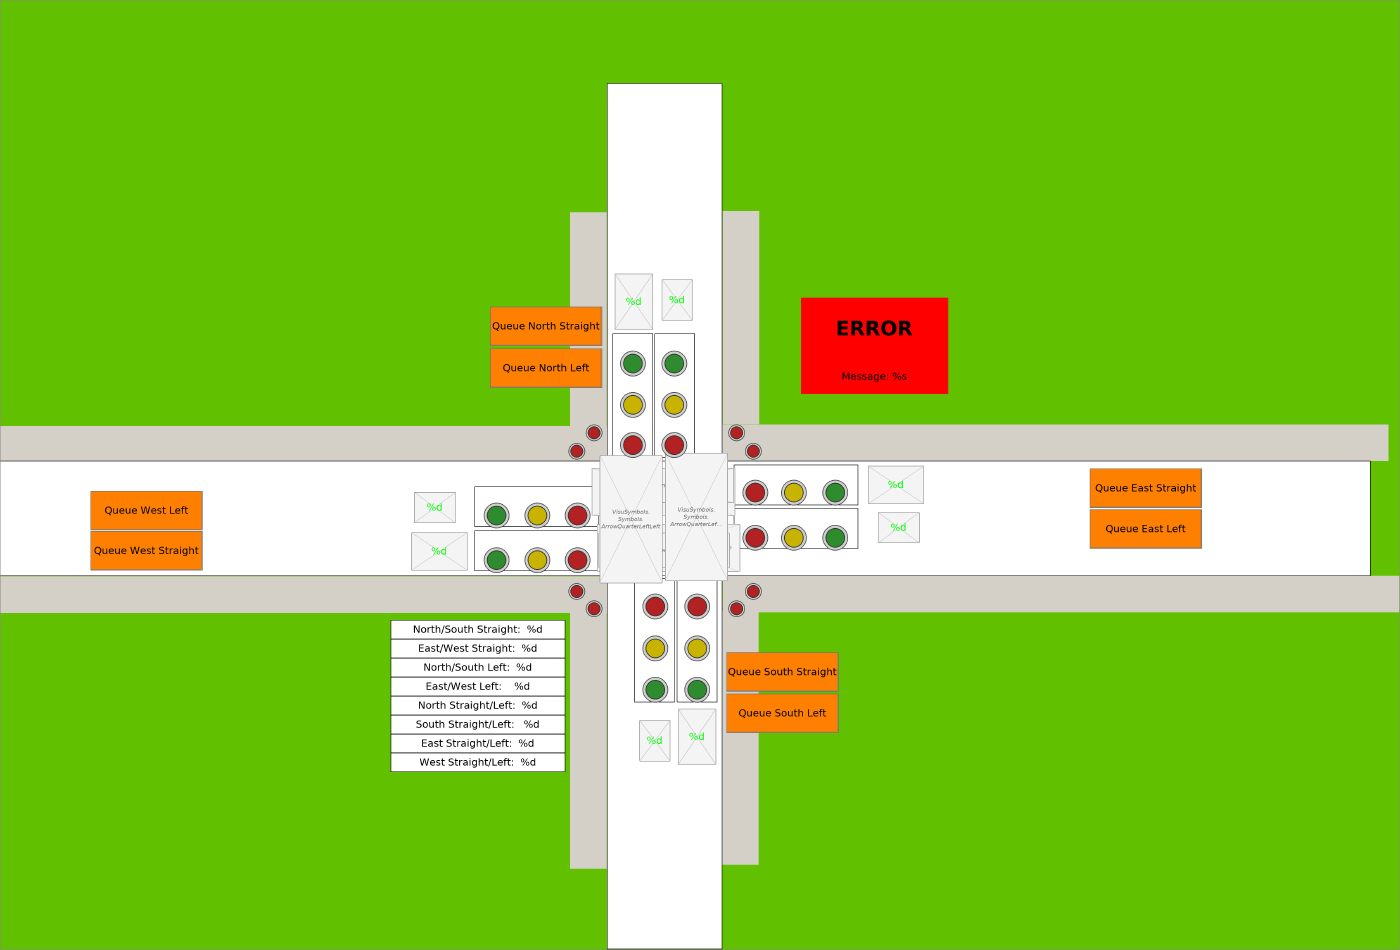
VISUALIZATION IntersectionVisual  // 2505x1701
    Rectangle (1292,1094 65x454)
    Rectangle (1020,1095 65x460)
    Rectangle (1020,380 65x384)
    Rectangle (1293,378 65x381)
    Rectangle (1293,1031 1210x65)
    Rectangle (0,1032 1088x65)
    Rectangle (0,763 1086x65)
    Rectangle (1291,760 1193x65)
    Rectangle (1086,149 206x1550)
    Rectangle (0,825 2452x206)
    Label (2086,901 197x64), "East"
    Label (1090,415 197x64), "North"
    Label (1091,1392 197x64), "South"
    Label (14,891 197x64), "West"
    RoundedRectangle (1313,832 222x72)
    Lamp1 (1394,840 53x84), variable: EastLight_Control.StraightYellowLight, style: Lamp-Lamp1-Yellow
    Lamp1 (1468,840 53x84), variable: EastLight_Control.StraightGreenLight, style: Lamp-Lamp1-Green
    Image (1553,834 100x68), "%d", text variable: Glbl.eastStraightSensorCnt, invisible if: NOT Glbl.eastStraightSensor, image: VisuSymbols.Symbols.ArrowBoldLeft
    RoundedRectangle (1313,910 222x72)
    Lamp1 (1394,921 53x84), variable: EastLight_Control.LeftYellowLight, style: Lamp-Lamp1-Yellow
    Lamp1 (1468,921 53x84), variable: EastLight_Control.LeftGreenLight, style: Lamp-Lamp1-Green
    Image (1571,917 74x55), "%d", text variable: Glbl.eastLeftSensorCnt, colour toggle: Glbl.eastLeftSensor, invisible if: Not Glbl.eastLeftSensor, image: VisuSymbols.Symbols.ArrowBoldDown
    Button (1950,839 200x70), "Queue East Straight"
        OnMouseDown: execute { Glbl.eastStraightSensor := TRUE; Glbl.eastStraightSensorCnt := Glbl.eastStraightSensorCnt + 1; }
    Button (1950,912 200x70), "Queue East Left"
        OnMouseDown: execute { Glbl.eastLeftSensor := TRUE; Glbl.eastLeftSensorCnt := Glbl.eastLeftSensorCnt + 1; }
    RoundedRectangle (849,871 222x72)
    RoundedRectangle (849,950 222x72)
    Lamp1 (1007,881 53x84), variable: WestLight_Control.LeftRedLight, style: Lamp-Lamp1-Red
    Lamp1 (935,881 53x84), variable: WestLight_Control.LeftYellowLight, style: Lamp-Lamp1-Yellow
    Lamp1 (862,881 53x84), variable: WestLight_Control.LeftGreenLight, style: Lamp-Lamp1-Green
    Lamp1 (1007,961 53x84), variable: WestLight_Control.StraightRedLight, style: Lamp-Lamp1-Red
    Lamp1 (935,961 53x84), variable: WestLight_Control.StraightYellowLight, style: Lamp-Lamp1-Yellow
    Lamp1 (862,961 53x84), variable: WestLight_Control.StraightGreenLight, style: Lamp-Lamp1-Green
    Image (736,953 100x68), "%d", text variable: Glbl.westStraightSensorCnt, invisible if: Not Glbl.westStraightSensor, image: VisuSymbols.Symbols.ArrowBoldRight
    Image (741,881 74x55), "%d", text variable: Glbl.westLeftSensorCnt, invisible if: Not Glbl.westLeftSensor, image: VisuSymbols.Symbols.ArrowBoldUp
    Button (162,951 200x70), "Queue West Straight"
        OnMouseDown: execute { Glbl.westStraightSensor := TRUE; Glbl.westStraightSensorCnt := Glbl.westStraightSensorCnt + 1; }
    Button (162,879 200x70), "Queue West Left"
        OnMouseDown: execute { Glbl.westLeftSensor := TRUE; Glbl.westLeftSensorCnt := Glbl.westLeftSensorCnt + 1; }
    Lamp1 (1301,1070 34x40), variable: SouthLight_Control.CrosswalkLight, invisible if: NOT SouthLight_Control.CrosswalkLight, style: Lamp-Lamp1-Green
    Lamp1 (1331,1039 34x40), variable: EastLight_Control.CrosswalkLight, invisible if: NOT EastLight_Control.CrosswalkLight, style: Lamp-Lamp1-Green
    Lamp1 (1046,1070 34x40), variable: SouthLight_Control.CrosswalkLight, invisible if: NOT SouthLight_Control.CrosswalkLight, style: Lamp-Lamp1-Green
    Lamp1 (1015,1039 34x40), variable: WestLight_Control.CrosswalkLight, invisible if: NOT WestLight_Control.CrosswalkLight, style: Lamp-Lamp1-Green
    Lamp1 (1331,788 34x40), variable: EastLight_Control.CrosswalkLight, invisible if: NOT EastLight_Control.CrosswalkLight, style: Lamp-Lamp1-Green
    Lamp1 (1301,755 34x40), variable: NorthLight_Control.CrosswalkLight, invisible if: NOT NorthLight_Control.CrosswalkLight, style: Lamp-Lamp1-Green
    Lamp1 (1015,788 34x40), variable: WestLight_Control.CrosswalkLight, invisible if: NOT WestLight_Control.CrosswalkLight, style: Lamp-Lamp1-Green
    Lamp1 (1046,755 34x40), variable: NorthLight_Control.CrosswalkLight, invisible if: NOT NorthLight_Control.CrosswalkLight, style: Lamp-Lamp1-Green
    Lamp1 (1331,788 34x40), variable: NOT EastLight_Control.CrosswalkLight, invisible if: EastLight_Control.CrosswalkLight, style: Lamp-Lamp1-Red
    Lamp1 (1301,755 34x40), variable: NOT NorthLight_Control.CrosswalkLight, invisible if: NorthLight_Control.CrosswalkLight, style: Lamp-Lamp1-Red
    Lamp1 (1331,1039 34x40), variable: NOT EastLight_Control.CrosswalkLight, invisible if: EastLight_Control.CrosswalkLight, style: Lamp-Lamp1-Red
    Lamp1 (1301,1070 34x40), variable: NOT SouthLight_Control.CrosswalkLight, invisible if: SouthLight_Control.CrosswalkLight, style: Lamp-Lamp1-Red
    Lamp1 (1046,755 34x40), variable: NOT NorthLight_Control.CrosswalkLight, invisible if: NorthLight_Control.CrosswalkLight, style: Lamp-Lamp1-Red
    Lamp1 (1015,788 34x40), variable: NOT WestLight_Control.CrosswalkLight, invisible if: WestLight_Control.CrosswalkLight, style: Lamp-Lamp1-Red
    Lamp1 (1015,1039 34x40), variable: NOT WestLight_Control.CrosswalkLight, invisible if: WestLight_Control.CrosswalkLight, style: Lamp-Lamp1-Red
    Lamp1 (1046,1070 34x40), variable: NOT SouthLight_Control.CrosswalkLight, invisible if: SouthLight_Control.CrosswalkLight, style: Lamp-Lamp1-Red
    Image (1059,838 256x85), invisible if: NOT Glbl.westLeftActive, image: VisuSymbols.Symbols.ArrowQuarterLeftUp
    Image (1068,938 256x85), invisible if: NOT Glbl.eastLeftActive, image: VisuSymbols.Symbols.ArrowQuarterLeftDown
    Image (1079,838 234x62), invisible if: NOT Glbl.eastStraightActive, image: VisuSymbols.Symbols.ArrowBoldLeft
    Image (1071,954 234x62), invisible if: Not Glbl.westStraightActive, image: VisuSymbols.Symbols.ArrowBoldRight
    RoundedRectangle (1211,1035 72x222)
    RoundedRectangle (1135,1035 72x222)
    Lamp1 (1221,1044 53x84), variable: SouthLight_Control.StraightRedLight, style: Lamp-Lamp1-Red
    Lamp1 (1146,1044 53x84), variable: SouthLight_Control.LeftRedLight, style: Lamp-Lamp1-Red
    Lamp1 (1146,1119 53x84), variable: SouthLight_Control.LeftYellowLight, style: Lamp-Lamp1-Yellow
    Lamp1 (1221,1119 53x84), variable: SouthLight_Control.StraightYellowLight, style: Lamp-Lamp1-Yellow
    Lamp1 (1146,1193 53x84), variable: SouthLight_Control.LeftGreenLight, style: Lamp-Lamp1-Green
    Lamp1 (1221,1193 53x84), variable: SouthLight_Control.StraightGreenLight, style: Lamp-Lamp1-Green
    Button (1300,1168 200x70), "Queue South Straight"
        OnMouseDown: execute { Glbl.southStraightSensor := TRUE; Glbl.southStraightSensorCnt := Glbl.southStraightSensorCnt + 1; }
    Button (1300,1242 200x70), "Queue South Left"
        OnMouseDown: execute { Glbl.southLeftSensor := TRUE; Glbl.southLeftSensorCnt := Glbl.southLeftSensorCnt + 1; }
    RoundedRectangle (1096,597 72x222)
    RoundedRectangle (1171,597 72x222)
    Image (1144,1289 55x74), "%d", text variable: Glbl.southLeftSensorCnt, invisible if: NOT Glbl.southLeftSensor, image: VisuSymbols.Symbols.ArrowBoldLeft
    Image (1213,1269 68x100), "%d", text variable: Glbl.southStraightSensorCnt, invisible if: Not Glbl.southStraightSensor, image: VisuSymbols.Symbols.ArrowBoldUp
    Image (1096,822 62x193), colour toggle: Glbl.eastLeftSensor, invisible if: Not Glbl.northStraightActive, image: VisuSymbols.Symbols.ArrowBoldDown
    Image (1215,841 62x193), invisible if: Not Glbl.southStraightActive, image: VisuSymbols.Symbols.ArrowBoldUp
    Image (1190,811 112x229), invisible if: NOT Glbl.northLeftActive, image: VisuSymbols.Symbols.ArrowQuarterLeftRight
    Image (1073,815 112x229), invisible if: NOT Glbl.southLeftActive, image: VisuSymbols.Symbols.ArrowQuarterLeftLeft
    Lamp1 (1106,755 53x84), variable: NorthLight_Control.StraightRedLight, style: Lamp-Lamp1-Red
    Lamp1 (1106,683 53x84), variable: NorthLight_Control.StraightYellowLight, style: Lamp-Lamp1-Yellow
    Lamp1 (1106,609 53x84), variable: NorthLight_Control.StraightGreenLight, style: Lamp-Lamp1-Green
    Lamp1 (1180,755 53x84), variable: NorthLight_Control.LeftRedLight, style: Lamp-Lamp1-Red
    Lamp1 (1180,683 53x84), variable: NorthLight_Control.LeftYellowLight, style: Lamp-Lamp1-Yellow
    Lamp1 (1180,609 53x84), variable: NorthLight_Control.LeftGreenLight, style: Lamp-Lamp1-Green
    Button (877,549 200x70), "Queue North Straight"
        OnMouseDown: execute { Glbl.northStraightSensor := TRUE; Glbl.northStraightSensorCnt := Glbl.northStraightSensorCnt + 1; }
    Button (877,624 200x70), "Queue North Left"
        OnMouseDown: execute { Glbl.northLeftSensor := TRUE; Glbl.northLeftSensorCnt := Glbl.northLeftSensorCnt + 1; }
    Image (1100,490 68x100), "%d", text variable: Glbl.northStraightSensorCnt, colour toggle: Glbl.eastLeftSensor, invisible if: Not Glbl.northStraightSensor, image: VisuSymbols.Symbols.ArrowBoldDown
    Image (1184,500 55x74), "%d", text variable: Glbl.northLeftSensorCnt, invisible if: Not Glbl.northLeftSensor, image: VisuSymbols.Symbols.ArrowBoldRight
    Lamp1 (1325,921 53x84), variable: EastLight_Control.leftRedLight, style: Lamp-Lamp1-Red
    Lamp1 (1325,840 53x84), variable: EastLight_Control.StraightRedLight, style: Lamp-Lamp1-Red
    Rectangle (699,1110 312x34), "North/South Straight: %d", text variable: Glbl.state1Counter
    Rectangle (699,1144 312x34), "East/West Straight: %d", text variable: Glbl.state2Counter
    Rectangle (699,1178 312x34), "North/South Left: %d", text variable: Glbl.state3Counter
    Rectangle (699,1212 312x34), "East/West Left: %d", text variable: Glbl.state4Counter
    Rectangle (699,1246 312x34), "North Straight/Left: %d", text variable: Glbl.state5Counter
    Rectangle (699,1280 312x34), "South Straight/Left: %d", text variable: Glbl.state6Counter
    Rectangle (699,1314 312x34), "East Straight/Left: %d", text variable: Glbl.state7Counter
    Rectangle (699,1348 312x34), "West Straight/Left: %d", text variable: Glbl.state8Counter
    Rectangle (1433,533 263x110), "ERROR", invisible if: NOT Glbl.error
    Rectangle (1433,643 263x62), "Message: %s", text variable: Glbl.errorMsg
END_VISUALIZATION

(* stored: Version 1.1.0.1, ProductVersion 3.1.4022.10
   Visu IntersectionVisual: Id {8b56e470-efa1-4cd6-9828-f0d17999d18f} *)
